// TwinCAT 3 PLC project EventTablePLC
// ProgramVersion: 3.1.4023.0
// libraries:
//   Tc2_Standard, * (Beckhoff Automation GmbH)
//   Tc2_System, * (Beckhoff Automation GmbH)
//   Tc2_Utilities, * (Beckhoff Automation GmbH)
//   Tc3_Module, * (Beckhoff Automation GmbH)
//   VisuSymbols,3.5.10.0,System
// project tree:
//   / GlobalTextList.TcGTLO, PlcTask.TcTTO, Visualization Manager.TcVMO (not stored), VISU_TASK.TcTTO
//   GVLs/GVLsEventsSimple/ GVL_EventsSimple.TcGVL
//   POUs/ MAIN.TcPOU
//   POUs/POUsEventsSimple/ FB_SimpleEventLog.TcPOU, P_EventsSimple.TcPOU
//   VISUs/ Visualization.TcVIS
// real-time tasks:
//   TASK PlcTask: cycle T#10ms, priority 20, ADS port 350
//   TASK VISU_TASK: cycle T#200000us, priority 30, ADS port 351

CONFIGURATION EventTablePLC
    RESOURCE PLC ON TwinCAT3
        TASK PlcTask(INTERVAL := T#10ms, PRIORITY := 20);
        TASK VISU_TASK(INTERVAL := T#200000us, PRIORITY := 30);
        PROGRAM MAIN WITH PlcTask : MAIN;
        PROGRAM VisuElems_Visu_Prg WITH VISU_TASK : VisuElems.Visu_Prg;
    END_RESOURCE
END_CONFIGURATION

// ---- GVLs/GVLsEventsSimple/GVL_EventsSimple.TcGVL
//==================================================================================================
//							Beckhoff Automation Poland
//									22.12.2016
//  v1.3	|| TC v 3.1.4020.28		|| - FIRST_MESSAGE i LAST_MESSAGE zmian typu z UDINT na DINT - znikaja ostrzezenia
//  v1.2	|| TC v 3.1.4020.28		|| - zmiana nazwy zakładki globalnych, zmiana nazwy zmiennej aAlarms na aEventsSimple
//  v1.1	|| TC v 3.1.4020.28		|| - dodanie wersjonowania: dodanie MSG_MESSAGE_List
// 	v1.0	|| TC v 3.1.4020.0		|| - pierwsza wersja
//==================================================================================================
VAR_GLOBAL CONSTANT
	FIRST_MESSAGE			: DINT := 1;
	LAST_MESSAGE			: DINT := 1200;
END_VAR
VAR_GLOBAL
	// Tablice alarmow, komunikatow i ostrzezen.
	MSG_ALARM_List			: ARRAY[FIRST_MESSAGE..LAST_MESSAGE] OF BOOL;
	MSG_WARNING_List		: ARRAY[FIRST_MESSAGE..LAST_MESSAGE] OF BOOL;
	MSG_MESSAGE_List		: ARRAY[FIRST_MESSAGE..LAST_MESSAGE] OF BOOL;
	aEventsSimple			: ARRAY[1..80] OF ST_ReadEvent;					// Tablica odczytywana przez obiekt wizualizacji Event table
	bAlarm					: BOOL;
	bWarning				: BOOL;
	bMessage				: BOOl;
END_VAR

// ---- POUs/MAIN.TcPOU
PROGRAM MAIN
VAR
END_VAR

P_EventsSimple();

END_PROGRAM

// ---- POUs/POUsEventsSimple/P_EventsSimple.TcPOU
//==================================================================================================
//							Beckhoff Automation Poland
//									5.2.2016
//		Program sluzy do przesylania globalnych tablic alarmow, ostrzezen i komunikatow do Event Loggera
//  v1.3	|| TC v 3.1.4020.28		|| - poprawki w MESSAGE, dodatkowe komentarze
//  v1.3	|| TC v 3.1.4020.28		|| - kosmetyka
//  v1.2	|| TC v 3.1.4020.28		|| - dodanie MESSAGE
//  v1.1 	|| TC v 3.1.4020.14 	|| - dodanie wersjonowania, komentarzy
// 	v1.0 	|| TC v 3.1.4020.0 		|| - pierwsza wersja
//==================================================================================================
PROGRAM P_EventsSimple
VAR
	fbAlarms				: FB_SimpleEventLog;								// Logowanie alarmow
	fbWarnings				: FB_SimpleEventLog;								// Logowanie ostrzezen
	fbMessage				: FB_SimpleEventLog;								// Logowanie komunikatow
	fbRead1					: FB_AdsReadEvents;									// Odczyt tablicy jezyk polski
	fbRead2					: FB_AdsReadEvents;									// Odczyt tablicy jezyk angielski
	fbRead3					: FB_AdsReadEvents;									// Odczyt tablicy jezyk niemiecki
	fbClear					: ADSCLEAREVENTS;									// Czyszczenie aktywnych alarmow
	MSG_ALARM_ListQuit		: ARRAY[FIRST_MESSAGE..LAST_MESSAGE] OF BOOL;		// Tablica nieuzywana - wymaga potwierdzenia przy usuwaniu
	MSG_MESSAGE_ListQuit	: ARRAY[FIRST_MESSAGE..LAST_MESSAGE] OF BOOL;		// Tablica nieuzywana - wymaga potwierdzenia przy usuwaniu
	MSG_WARNING_ListQuit	: ARRAY[FIRST_MESSAGE..LAST_MESSAGE] OF BOOL;		// Tablica nieuzywana - wymaga potwierdzenia przy usuwaniu
END_VAR

(*
	TCEVENTCLASS_NONE			:=0,	No class
	TCEVENTCLASS_MAINTENANCE	:=1,	Maintenance hint
	TCEVENTCLASS_MESSAGE		:=2,	Message
	TCEVENTCLASS_HINT			:=3,	Hint
	TCEVENTCLASS_STATEINFO		:=4,	State information
	TCEVENTCLASS_INSTRUCTION	:=5,	Instruction
	TCEVENTCLASS_WARNING		:=6,	Warning
	TCEVENTCLASS_ALARM			:=7,	Alarm
	TCEVENTCLASS_PARAMERROR		:=8	 	Parameter error
*)
A_Active();
fbClear(	bClear			:= TRUE,
			iMode			:= TCEVENTLOGIOFFS_CLEARALL);

fbAlarms(	Init			:= TRUE,
			SourceId		:= 1,
			Class			:= TCEVENTCLASS_ALARM,
			QuitRequired	:= FALSE,
			adrAlarmArray	:= ADR(MSG_ALARM_List),
			adrQuitArray	:= ADR(MSG_ALARM_ListQuit));
	
fbWarnings(	Init			:= TRUE,
			SourceId		:= 2,
			Class			:= TCEVENTCLASS_WARNING,
			QuitRequired	:= FALSE,
			adrAlarmArray	:= ADR(MSG_WARNING_List),
			adrQuitArray	:= ADR(MSG_WARNING_ListQuit));

fbMessage(	Init			:= TRUE,
			SourceId		:= 3,
			Class			:= TCEVENTCLASS_MESSAGE,
			QuitRequired	:= FALSE,
			adrAlarmArray	:= ADR(MSG_MESSAGE_List),
			adrQuitArray	:= ADR(MSG_MESSAGE_ListQuit));
			
// Odczyt w kilku jezykach
fbRead1(	bReadEvents		:= TRUE,
			nLanguageId		:= 1045,
			tRefreshTime	:= T#1S);

fbRead2(	bReadEvents		:= TRUE,
			nLanguageId		:= 1033,
			tRefreshTime	:= T#1S);

fbRead3(	bReadEvents		:= TRUE, 
			nLanguageId		:= 1031, 
			tRefreshTime	:= T#1S);
			
// Wybor aktualnego jezyka wyswietlania - przepisanie do tablicy odpowiedniej tablicy
// Uwaga j. polski bez polskich znakow
IF VisuElemsWinControls.CURRENTLANGUAGE		= 'en' THEN
	aEventsSimple			:= fbRead2.aEvents;
ELSIF VisuElemsWinControls.CURRENTLANGUAGE	= 'de' THEN
	aEventsSimple			:= fbRead3.aEvents;
ELSE
	aEventsSimple			:= fbRead1.aEvents;	
END_IF;

ACTION A_Active:
GVL_EventsSimple.MSG_ALARM_List[1]:=GVL_EventsSimple.bAlarm;
GVL_EventsSimple.MSG_WARNING_List[1]:=GVL_EventsSimple.bWarning;
GVL_EventsSimple.MSG_MESSAGE_List[1]:=GVL_EventsSimple.bMessage;
END_ACTION

END_PROGRAM

// ---- POUs/POUsEventsSimple/FB_SimpleEventLog.TcPOU
//==================================================================================================
//							Beckhoff Automation Poland
//									22.12.2016
//	Program glowny dla zdarzen wersji advanced
// 	v1.1	|| TC v 3.1.4020.28		|| - idx, ARRAY_LBOUND, ARRAY_UBOUND --> Zmiana typu z UDINT na DINT
// 	v1.0	|| TC v 3.1.4020.28		|| - pierwsza wersja - 13.10.2004, Author:			Dirk Nordberg (BECKHOFF INDUSTRIE ELEKTRONIK)
// Description: Function block to control the EventLogger
// 	Messages can be activated or deactivated through an array of bool.
// 	The subscription of the array is equivalent to EventID from EventLogger.
// 	Funtion block will be initialized with Init flag, then the busy flag is set true. 
// 
// 	Revision:	1.4
// 	History:		13.10.2004	Ng	start coding
// 					17.04.2005	MK	runtime optimized
// 					07.07.2005	MK	short puls BF
// 				    29.11.2010 	MiB  quittierungspflichtige Merker funktionieren nun wieder
///                 21.06.2013  TV   change : data type for pointer address from uint to pointer of int 
//==================================================================================================
///****************************************************************************************
///Name:				FB_SimpleEventLog
///Date:				13.10.2004
// 

FUNCTION_BLOCK FB_SimpleEventLog
VAR_INPUT
	/// Rising flag starts the initialization 
	Init: BOOL;
	/// Number of the source Id 
	SourceId: UINT;
	/// Alarm error class 
	Class: UINT;
	/// Activate or deaktivate confirmation 
	QuitRequired: BOOL;
	/// Adress of the array for the messages 
	adrAlarmArray: POINTER TO BOOL;
	/// ...with constant boundaries ARRAY_LBOUND to ARRAY_UBOUND for array size 
	adrQuitArray: POINTER TO BOOL;
END_VAR
VAR_OUTPUT
	Busy: BOOL;
	Err: BOOL;
	ErrId: UDINT;
END_VAR
VAR CONSTANT
	ARRAY_LBOUND: DINT := FIRST_MESSAGE;
	ARRAY_UBOUND: DINT := LAST_MESSAGE;
	TCEVENTDATAFORMATSTRING: STRING := ' ';
	STATE_INIT: INT := 0;
	STATE_IDLE: INT := 1;
	STATE_RESET_EVENT: INT := 2;
	STATE_QUIT_EVENT: INT := 3;
	STATE_RESET_END: INT := 4;
	STATE_WAIT: INT := 5;
END_VAR
VAR
	state: INT;
	///{flag nowatch on }
	bReady: BOOL := TRUE;
	nMsgHasChanged: DINT;
	bEvtState: ARRAY[ARRAY_LBOUND..ARRAY_UBOUND] OF BOOL;
	event: ARRAY[ARRAY_LBOUND..ARRAY_UBOUND] OF ADSLOGEVENT;
	idx: DINT;
	CfgEvent: TcEvent;
	bWait: BOOL;
	ptAlarm: POINTER TO BOOL;
	ptQuit: POINTER TO BOOL;
	RT_Init: R_TRIG;
END_VAR

nMsgHasChanged := MEMCMP(ADR(bEvtState), adrAlarmArray, SIZEOF(bEvtState));

RT_Init(CLK:=Init);

CASE State OF
	STATE_INIT:		(* Set the parameter for TcEvent *)
		Err := FALSE;
		ErrId :=0;
		Busy := FALSE;
		CfgEvent.Prio := 0;
		CfgEvent.DataFormatStrAddress := ADR(TCEVENTDATAFORMATSTRING);
		// CfgEvent.Flags := TCEVENTFLAG_LOG OR TCEVENTFLAG_SRCID OR TCEVENTFLAG_PRIOCLASS OR TCEVENTFLAG_FMTSELF OR 16#1000;
		// MiB 2015.10.07 Flags changed -> now the class is defined here and not in Event config file.
		CfgEvent.Flags := TCEVENTFLAG_LOG OR TCEVENTFLAG_SRCID;
		CfgEvent.StreamType := TCEVENTSTREAM_SIMPLE;
		CfgEvent.ProgId := 'TcEventFormatter.TcXmlFormatter';
		CfgEvent.SourceId := SourceId;
			CfgEvent.Class := Class ;
		CfgEvent.bQuitRequired := QuitRequired;
		FOR idx := ARRAY_LBOUND TO ARRAY_UBOUND BY 1 DO
			CfgEvent.Id := DINT_TO_UDINT(idx);
			event[idx](NETID:='', PORT:=110, Event:=FALSE , EventQuit:=FALSE,
				 EventConfigData:=CfgEvent, FbCleanup:=FALSE, TMOUT:=t#1s);
		END_FOR;
		State := STATE_IDLE;

	STATE_IDLE:
		(* nothing to do *)
		IF nMsgHasChanged = 0
			AND  NOT QuitRequired
			AND bReady = TRUE
			AND NOT RT_Init.Q THEN
			RETURN;
		END_IF

		IF adrAlarmArray <> 0 THEN
			ptAlarm := adrAlarmArray;
			IF CfgEvent.bQuitRequired AND adrQuitArray <> 0 THEN
				ptQuit := adrQuitArray;
				FOR idx := ARRAY_LBOUND TO ARRAY_UBOUND BY 1 DO
					event[idx](Event:=ptAlarm^, EventQuit:=ptQuit^);
					ptAlarm := ptAlarm + 1;
					ptQuit := ptQuit + 1;
				END_FOR;
				bReady := TRUE;
			ELSE
				bReady := TRUE;
				FOR idx := ARRAY_LBOUND TO ARRAY_UBOUND BY 1 DO
					event[idx](Event:=ptAlarm^);
					IF (NOT (ptAlarm^ = TRUE
							AND event[idx].Event = TRUE		(* event is set/on *)
							AND event[idx].Quit = FALSE
							AND event[idx].EventState = TCEVENTSTATE_SIGNALED)
						AND NOT (ptAlarm^ = FALSE
							AND event[idx].Event = FALSE		(* event is reset/off *)
							AND event[idx].Quit = TRUE
							AND event[idx].EventState = TCEVENTSTATE_INVALID)) THEN
						bReady := FALSE;
					END_IF
					ptAlarm := ptAlarm + 1;
				END_FOR;

				(* copy the status *)
				IF bReady THEN
					MEMCPY(ADR(bEvtState), adrAlarmArray, SIZEOF(bEvtState));
				END_IF

			END_IF
		END_IF

		IF RT_Init.Q THEN
			Busy := TRUE;
			State := STATE_RESET_EVENT;
		END_IF

	STATE_RESET_EVENT:(*---------------------------------- clear messages ----------------------------------------*)
		FOR idx := ARRAY_LBOUND TO ARRAY_UBOUND BY 1 DO
			IF event[idx].EventState = TCEVENTSTATE_SIGNALED THEN
				event[idx](Event:=FALSE, EventQuit:= FALSE, FbCleanup:= FALSE, TMOUT:= t#1s);
				IF event[idx].Err THEN
					Err := TRUE;
					ErrId := event[idx].ErrId;
					IF event[idx].ErrId = 1282 THEN	(* Message Router: mailbox full *)
						event[idx](Event:=FALSE, EventQuit:= FALSE, FbCleanup:= FALSE);
						RETURN;
					END_IF
				END_IF
			END_IF;
		END_FOR;
		State := STATE_QUIT_EVENT;

	STATE_QUIT_EVENT:(*---------------------------------- quit messages ----------------------------------------*)
		FOR idx := ARRAY_LBOUND TO ARRAY_UBOUND BY 1 DO
			IF event[idx].EventState = TCEVENTSTATE_SIGNALED THEN
				event[idx](Event:=FALSE, EventQuit:= TRUE, FbCleanup:= FALSE, TMOUT:= t#1s);
				IF event[idx].Err THEN
					Err := TRUE;
					ErrId := event[idx].ErrId;
					IF event[idx].ErrId = 1282 THEN	(* Message Router: mailbox full *)
						event[idx](Event:=FALSE, EventQuit:= FALSE, FbCleanup:= FALSE);
						RETURN;
					END_IF
				END_IF
			END_IF;
		END_FOR;
		State := STATE_RESET_END;

	STATE_RESET_END:
		bWait := FALSE;
		FOR idx := ARRAY_LBOUND TO ARRAY_UBOUND BY 1 DO
			event[idx](Event:=FALSE, EventQuit:= FALSE, FbCleanup:= FALSE);
			IF event[idx].EventState = TCEVENTSTATE_SIGNALED THEN
				bWait := TRUE;
			END_IF
		END_FOR;
		IF NOT bWait THEN
			State := STATE_INIT;
		END_IF

END_CASE

END_FUNCTION_BLOCK

// ---- VISUs/Visualization.TcVIS
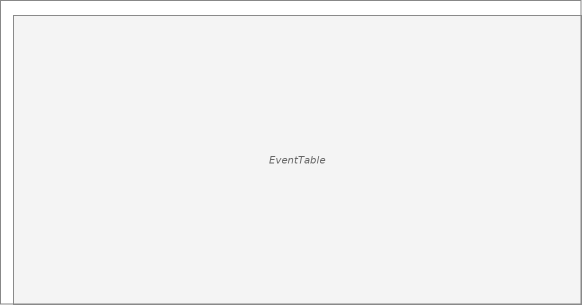
VISUALIZATION Visualization  // 582x305
    EventTable (13,15 569x290)
        p1690906150: Class
        p3258520714: Date
        p2231227367: Time
        p3993844394: Message
        p2076579579: Details
        p3558512729: GVL_EventsSimple.aEventsSimple
        p3921149237: m_pDataArray..pArray
END_VISUALIZATION
